PROGRAM MAIN
VAR
END_VAR

END_PROGRAM

(* stored: Version 1.1.0.1
   POU MAIN: Id {4c7ef0bc-b25c-464c-94d8-383fa37d5736} *)
